FUNCTION_BLOCK FB_SYS_DT (* Request the system date and time *)
  (* Standard: 61499-2 *)
  (* Version 1.0, 2017-09-05, Marc Jakobi, HTW Berlin *)
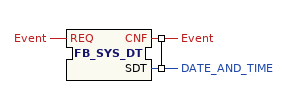
  EVENT_INPUT
    REQ; (* Service Request *)
  END_EVENT
  EVENT_OUTPUT
    CNF WITH SDT; (* Confirmation of Requested Service *)
  END_EVENT
  VAR_OUTPUT
    SDT : DATE_AND_TIME; (* System date and time *)
  END_VAR
  (* Service APPLICATION/RESOURCE: Request the system date and time *)
END_FUNCTION_BLOCK
